TYPE ProgrammaLog :
STRUCT
	Programma : ARRAY[0..10] OF Descrittore_Programma;
END_STRUCT
END_TYPE

(* stored: Version 1.1.0.1, ProductVersion 3.1.4024.11
   DUT ProgrammaLog: Id {5cb04c68-2afc-4306-b264-cd2b43f7b71b} *)
